(* IEC 61131-3 sources: Std_PalletMover/Class/_ComDiagnosis, 1 file *)

(* ---- _ComDiagnosis.st ---- *)
#define COMDIAG_COMMAND                 (10000)
#define COMDIAG_MAJORID_COMDIAGNOSIS    (10003)
#define COMDIAG_MINORID_CMDRESETDIAGS   (0)
#define COMDIAG_MINORID_CONNECTCNT      (1)
#define COMDIAG_MINORID_CONNECTFAILCNT  (2)
#define COMDIAG_MINORID_RETRYCNT        (3)
#define COMDIAG_MINORID_WATCHDOGCNT     (4)
#define COMDIAG_MINORID_ACTERRORCODE    (5)
#define COMDIAG_MINORID_LASTERRORCODE   (6)
#define COMDIAG_MINORID_ERRORCNT        (7)
#define COMDIAG_MINORID_READCNT         (8)
#define COMDIAG_MINORID_READERRORCNT    (9)
#define COMDIAG_MINORID_WRITECNT        (10)
#define COMDIAG_MINORID_WRITEERRORCNT   (11)

(*!
<Class
	Name               = "_ComDiagnosis"
	Revision           = "1.0"
	RealtimeTask       = "false"
	CyclicTask         = "false"
	BackgroundTask     = "true"
	DefBackground      = "50 ms"
	Sigmatek           = "true"
	OSInterface        = "false"
	HighPriority       = "false"
	Automatic          = "false"
	UpdateMode         = "Prescan"
	SharedCommandTable = "true"
	Objectsize         = "(496,120)"
	Comment            = "This class display and forwards diagnosis information on communication.">
	<Channels>
		<Server Name="ActErrorCode" Visualized="false" Initialize="false" WriteProtected="true" Retentive="false" Comment="Actual error code of connected ComObject - Read is called every cycle."/>
		<Server Name="ClassSvr" Visualized="false" Initialize="false" WriteProtected="true" Retentive="false"/>
		<Server Name="CmdResetDiags" Visualized="true" Initialize="false" WriteProtected="false" Retentive="false" Comment="Class with a write method, that resets all counter values. DINT"/>
		<Server Name="ConnectCnt" Visualized="false" Initialize="false" WriteProtected="true" Retentive="false" Comment="Number of Connect Attempts - Read is called every cycle."/>
		<Server Name="ConnectFailCnt" Visualized="false" Initialize="false" WriteProtected="true" Retentive="false" Comment="Number of Connect Failures - Read is called every cycle."/>
		<Server Name="ErrorCnt" Visualized="false" Initialize="false" WriteProtected="true" Retentive="false" Comment="Number of Errors - Read is called every cycle."/>
		<Server Name="LastErrorCode" Visualized="false" Initialize="false" WriteProtected="true" Retentive="false" Comment="Last error code of connected ComObject - Read is called every cycle."/>
		<Server Name="ReadCnt" Visualized="false" Initialize="false" WriteProtected="true" Retentive="false" Comment="Number of Reads - Read is called every cycle."/>
		<Server Name="ReadErrorCnt" Visualized="false" Initialize="false" WriteProtected="true" Retentive="false" Comment="Number of Read Errors - Read is called every cycle."/>
		<Server Name="RefreshCnt" Visualized="false" Initialize="false" WriteProtected="true" Retentive="false" Comment="Server that increments with every cycle."/>
		<Server Name="RetryCnt" Visualized="false" Initialize="false" WriteProtected="true" Retentive="false" Comment="Number of Connect Retries - Read is called every cycle."/>
		<Server Name="WatchdogCnt" Visualized="false" Initialize="false" WriteProtected="true" Retentive="false" Comment="Number of Watchdog Timeouts - Read is called every cycle."/>
		<Server Name="WriteCnt" Visualized="false" Initialize="false" WriteProtected="true" Retentive="false" Comment="Number of Writes - Read is called every cycle."/>
		<Server Name="WriteErrorCnt" Visualized="false" Initialize="false" WriteProtected="true" Retentive="false" Comment="Number of Write Errors - Read is called every cycle."/>
		<Client Name="ComObject" Required="false" Internal="false" Comment="CommandChannel which will be connected to the object to be diagnosed."/>
	</Channels>
	<Separators>
		<Servers>
			<SepChn Position="2"/>
			<SepChn Position="14"/>
		</Servers>
	</Separators>
	<RevDoku>
		<Owner Company="Sigmatek" Author="ZilSal"/>
		<Dokumentation Revision="1.0" Date="2019-04-10" Author="VelGer" Company="Sigmatek" Description="Optimization of Class."/>
		<Dokumentation Revision="0.9" Date="2019-03-08" Author="ZilSal" Company="Sigmatek" Description="Initial Creation of Class."/>
	</RevDoku>
</Class>
*)
_ComDiagnosis : CLASS
  //Servers:
	ClassSvr 	: SvrChCmd_DINT;
	RefreshCnt 	: SvrCh_DINT;
	ConnectCnt 	: SvrCh_DINT;
	ConnectFailCnt 	: SvrCh_DINT;
	RetryCnt 	: SvrCh_DINT;
	WatchdogCnt 	: SvrCh_DINT;
	ActErrorCode 	: SvrCh_DINT;
	LastErrorCode 	: SvrCh_DINT;
	ErrorCnt 	: SvrCh_DINT;
	ReadCnt 	: SvrCh_DINT;
	ReadErrorCnt 	: SvrCh_DINT;
	WriteCnt 	: SvrCh_DINT;
	WriteErrorCnt 	: SvrCh_DINT;
	CmdResetDiags 	: SvrCh_DINT;
  //Clients:
	ComObject 	: CltChCmd_DINT;
  //Variables:
  //Functions:

	FUNCTION VIRTUAL GLOBAL Background
		VAR_INPUT
			EAX 	: UDINT;
		END_VAR
		VAR_OUTPUT
			state (EAX) 	: UDINT;
		END_VAR;

	FUNCTION VIRTUAL GLOBAL RefreshCnt::Read
		VAR_OUTPUT
			output (EAX) 	: DINT;
		END_VAR;

	FUNCTION VIRTUAL GLOBAL ConnectCnt::Read
		VAR_OUTPUT
			output (EAX) 	: DINT;
		END_VAR;

	FUNCTION VIRTUAL GLOBAL ConnectFailCnt::Read
		VAR_OUTPUT
			output (EAX) 	: DINT;
		END_VAR;

	FUNCTION VIRTUAL GLOBAL RetryCnt::Read
		VAR_OUTPUT
			output (EAX) 	: DINT;
		END_VAR;

	FUNCTION VIRTUAL GLOBAL WatchdogCnt::Read
		VAR_OUTPUT
			output (EAX) 	: DINT;
		END_VAR;

	FUNCTION VIRTUAL GLOBAL ActErrorCode::Read
		VAR_OUTPUT
			output (EAX) 	: DINT;
		END_VAR;

	FUNCTION VIRTUAL GLOBAL LastErrorCode::Read
		VAR_OUTPUT
			output (EAX) 	: DINT;
		END_VAR;

	FUNCTION VIRTUAL GLOBAL ErrorCnt::Read
		VAR_OUTPUT
			output (EAX) 	: DINT;
		END_VAR;

	FUNCTION VIRTUAL GLOBAL ReadCnt::Read
		VAR_OUTPUT
			output (EAX) 	: DINT;
		END_VAR;

	FUNCTION VIRTUAL GLOBAL ReadErrorCnt::Read
		VAR_OUTPUT
			output (EAX) 	: DINT;
		END_VAR;

	FUNCTION VIRTUAL GLOBAL WriteCnt::Read
		VAR_OUTPUT
			output (EAX) 	: DINT;
		END_VAR;

	FUNCTION VIRTUAL GLOBAL WriteErrorCnt::Read
		VAR_OUTPUT
			output (EAX) 	: DINT;
		END_VAR;

	FUNCTION VIRTUAL GLOBAL CmdResetDiags::Write
		VAR_INPUT
			input (EAX) 	: DINT;
		END_VAR
		VAR_OUTPUT
			result (EAX) 	: DINT;
		END_VAR;
  //Tables:
	FUNCTION @STD
		VAR_OUTPUT
			ret_code	: CONFSTATES;
		END_VAR;
	FUNCTION GLOBAL TAB @CT_;
END_CLASS;

FUNCTION VIRTUAL GLOBAL _ComDiagnosis::Background
	VAR_INPUT
		EAX 	: UDINT;
	END_VAR
	VAR_OUTPUT
		state (EAX) 	: UDINT;
	END_VAR

  // Call all read methods
  ConnectCnt.Read();
  ConnectFailCnt.Read();
  RetryCnt.Read();
  WatchdogCnt.Read();
  ActErrorCode.Read();
  LastErrorCode.Read();
  ErrorCnt.Read();
  ReadCnt.Read();
  ReadErrorCnt.Read();
  WriteCnt.Read();
  WriteErrorCnt.Read();

  // Increment the refresh counter
  RefreshCnt += 1;

	state := READY;

END_FUNCTION

FUNCTION VIRTUAL GLOBAL _ComDiagnosis::RefreshCnt::Read
	VAR_OUTPUT
		output (EAX) 	: DINT;
	END_VAR

	output := RefreshCnt;

END_FUNCTION

FUNCTION VIRTUAL GLOBAL _ComDiagnosis::ConnectCnt::Read
	VAR_OUTPUT
		output (EAX) 	: DINT;
	END_VAR
  VAR
  	NiGive : CmdStruct;
    NiGet : results;
  END_VAR

  NiGive.uiCmd    := COMDIAG_COMMAND;
  NiGive.aPara[0] := COMDIAG_MAJORID_COMDIAGNOSIS;
  NiGive.aPara[1] := COMDIAG_MINORID_CONNECTCNT;

  _memset(dest:=#NiGet, usByte:=0, cntr:=sizeof(NiGet));

  ComObject.NewInst(#NiGive, #NiGet);

  ConnectCnt := NiGet.aData[0];

	output := ConnectCnt;

END_FUNCTION

FUNCTION VIRTUAL GLOBAL _ComDiagnosis::ConnectFailCnt::Read
	VAR_OUTPUT
		output (EAX) 	: DINT;
	END_VAR
  VAR
  	NiGive : CmdStruct;
    NiGet : results;
  END_VAR

  NiGive.uiCmd    := COMDIAG_COMMAND;
  NiGive.aPara[0] := COMDIAG_MAJORID_COMDIAGNOSIS;
  NiGive.aPara[1] := COMDIAG_MINORID_CONNECTFAILCNT;

  _memset(dest:=#NiGet, usByte:=0, cntr:=sizeof(NiGet));

  ComObject.NewInst(#NiGive, #NiGet);

  ConnectFailCnt := NiGet.aData[0];

	output := ConnectFailCnt;

END_FUNCTION

FUNCTION VIRTUAL GLOBAL _ComDiagnosis::RetryCnt::Read
	VAR_OUTPUT
		output (EAX) 	: DINT;
	END_VAR
  VAR
  	NiGive : CmdStruct;
    NiGet : results;
  END_VAR

  NiGive.uiCmd    := COMDIAG_COMMAND;
  NiGive.aPara[0] := COMDIAG_MAJORID_COMDIAGNOSIS;
  NiGive.aPara[1] := COMDIAG_MINORID_RETRYCNT;

  _memset(dest:=#NiGet, usByte:=0, cntr:=sizeof(NiGet));

  ComObject.NewInst(#NiGive, #NiGet);

  RetryCnt := NiGet.aData[0];

	output := RetryCnt;

END_FUNCTION

FUNCTION VIRTUAL GLOBAL _ComDiagnosis::WatchdogCnt::Read
	VAR_OUTPUT
		output (EAX) 	: DINT;
	END_VAR
  VAR
  	NiGive : CmdStruct;
    NiGet : results;
  END_VAR

  NiGive.uiCmd    := COMDIAG_COMMAND;
  NiGive.aPara[0] := COMDIAG_MAJORID_COMDIAGNOSIS;
  NiGive.aPara[1] := COMDIAG_MINORID_WATCHDOGCNT;

  _memset(dest:=#NiGet, usByte:=0, cntr:=sizeof(NiGet));

  ComObject.NewInst(#NiGive, #NiGet);

  WatchdogCnt := NiGet.aData[0];

	output := WatchdogCnt;

END_FUNCTION

FUNCTION VIRTUAL GLOBAL _ComDiagnosis::ActErrorCode::Read
	VAR_OUTPUT
		output (EAX) 	: DINT;
	END_VAR
  VAR
  	NiGive : CmdStruct;
    NiGet : results;
  END_VAR

  NiGive.uiCmd    := COMDIAG_COMMAND;
  NiGive.aPara[0] := COMDIAG_MAJORID_COMDIAGNOSIS;
  NiGive.aPara[1] := COMDIAG_MINORID_ACTERRORCODE;

  _memset(dest:=#NiGet, usByte:=0, cntr:=sizeof(NiGet));

  ComObject.NewInst(#NiGive, #NiGet);

  ActErrorCode := NiGet.aData[0];

	output := ActErrorCode;

END_FUNCTION

FUNCTION VIRTUAL GLOBAL _ComDiagnosis::LastErrorCode::Read
	VAR_OUTPUT
		output (EAX) 	: DINT;
	END_VAR
  VAR
  	NiGive : CmdStruct;
    NiGet : results;
  END_VAR

  NiGive.uiCmd    := COMDIAG_COMMAND;
  NiGive.aPara[0] := COMDIAG_MAJORID_COMDIAGNOSIS;
  NiGive.aPara[1] := COMDIAG_MINORID_LASTERRORCODE;

  _memset(dest:=#NiGet, usByte:=0, cntr:=sizeof(NiGet));

  ComObject.NewInst(#NiGive, #NiGet);

  LastErrorCode := NiGet.aData[0];

	output := LastErrorCode;

END_FUNCTION

FUNCTION VIRTUAL GLOBAL _ComDiagnosis::ErrorCnt::Read
	VAR_OUTPUT
		output (EAX) 	: DINT;
	END_VAR
  VAR
  	NiGive : CmdStruct;
    NiGet : results;
  END_VAR

  NiGive.uiCmd    := COMDIAG_COMMAND;
  NiGive.aPara[0] := COMDIAG_MAJORID_COMDIAGNOSIS;
  NiGive.aPara[1] := COMDIAG_MINORID_ERRORCNT;

  _memset(dest:=#NiGet, usByte:=0, cntr:=sizeof(NiGet));

  ComObject.NewInst(#NiGive, #NiGet);

  ErrorCnt := NiGet.aData[0];

	output := ErrorCnt;

END_FUNCTION

FUNCTION VIRTUAL GLOBAL _ComDiagnosis::ReadCnt::Read
	VAR_OUTPUT
		output (EAX) 	: DINT;
	END_VAR
  VAR
  	NiGive : CmdStruct;
    NiGet : results;
  END_VAR

  NiGive.uiCmd    := COMDIAG_COMMAND;
  NiGive.aPara[0] := COMDIAG_MAJORID_COMDIAGNOSIS;
  NiGive.aPara[1] := COMDIAG_MINORID_READCNT;

  _memset(dest:=#NiGet, usByte:=0, cntr:=sizeof(NiGet));

  ComObject.NewInst(#NiGive, #NiGet);

  ReadCnt := NiGet.aData[0];

	output := ReadCnt;

END_FUNCTION

FUNCTION VIRTUAL GLOBAL _ComDiagnosis::ReadErrorCnt::Read
	VAR_OUTPUT
		output (EAX) 	: DINT;
	END_VAR
  VAR
  	NiGive : CmdStruct;
    NiGet : results;
  END_VAR

  NiGive.uiCmd    := COMDIAG_COMMAND;
  NiGive.aPara[0] := COMDIAG_MAJORID_COMDIAGNOSIS;
  NiGive.aPara[1] := COMDIAG_MINORID_READERRORCNT;

  _memset(dest:=#NiGet, usByte:=0, cntr:=sizeof(NiGet));

  ComObject.NewInst(#NiGive, #NiGet);

  ReadErrorCnt := NiGet.aData[0];

	output := ReadErrorCnt;

END_FUNCTION

FUNCTION VIRTUAL GLOBAL _ComDiagnosis::WriteCnt::Read
	VAR_OUTPUT
		output (EAX) 	: DINT;
	END_VAR
  VAR
  	NiGive : CmdStruct;
    NiGet : results;
  END_VAR

  NiGive.uiCmd    := COMDIAG_COMMAND;
  NiGive.aPara[0] := COMDIAG_MAJORID_COMDIAGNOSIS;
  NiGive.aPara[1] := COMDIAG_MINORID_WRITECNT;

  _memset(dest:=#NiGet, usByte:=0, cntr:=sizeof(NiGet));

  ComObject.NewInst(#NiGive, #NiGet);

  WriteCnt := NiGet.aData[0];

	output := WriteCnt;

END_FUNCTION

FUNCTION VIRTUAL GLOBAL _ComDiagnosis::WriteErrorCnt::Read
	VAR_OUTPUT
		output (EAX) 	: DINT;
	END_VAR
  VAR
  	NiGive : CmdStruct;
    NiGet : results;
  END_VAR

  NiGive.uiCmd    := COMDIAG_COMMAND;
  NiGive.aPara[0] := COMDIAG_MAJORID_COMDIAGNOSIS;
  NiGive.aPara[1] := COMDIAG_MINORID_WRITEERRORCNT;

  _memset(dest:=#NiGet, usByte:=0, cntr:=sizeof(NiGet));

  ComObject.NewInst(#NiGive, #NiGet);

  WriteErrorCnt := NiGet.aData[0];

	output := WriteErrorCnt;

END_FUNCTION

FUNCTION VIRTUAL GLOBAL _ComDiagnosis::CmdResetDiags::Write
	VAR_INPUT
		input (EAX) 	: DINT;
	END_VAR
	VAR_OUTPUT
		result (EAX) 	: DINT;
	END_VAR
  VAR
  	NiGive : CmdStruct;
    NiGet : results;
  END_VAR

	CmdResetDiags := input;

  NiGive.uiCmd    := COMDIAG_COMMAND;
  NiGive.aPara[0] := COMDIAG_MAJORID_COMDIAGNOSIS;
  NiGive.aPara[1] := COMDIAG_MINORID_CMDRESETDIAGS;

  _memset(dest:=#NiGet, usByte:=0, cntr:=sizeof(NiGet));

  ComObject.NewInst(#NiGive, #NiGet);

  CmdResetDiags := 0;

	result := CmdResetDiags;

END_FUNCTION
